// TIA Portal project "durum_grafigi_1" (V18)

(* hardware
DEVICE "S7-1200 station_1"  S7-1200 Station
   slot 0: "Rack_0"  S7-1200 Rack  Rack  V1.0
   slot 1: "PLC_1"  CPU 1214C DC/DC/DC  6ES7 214-1AG40-0XB0  V4.6
*)

// ===== PLC "PLC_1"  CPU 1214C DC/DC/DC =====

VAR_GLOBAL   // PLC tag table "Default tag table"
   "BAŞLAT" AT %I0.0 : Bool;
   "seviye_1_S1" AT %I0.1 : Bool;
   "seviye_2_S2" AT %I0.2 : Bool;
   "seviye_3_S3" AT %I0.3 : Bool;
   "ısı_sensoru_S4" AT %I0.4 : Bool;
   "valf_1" AT %Q0.1 : Bool;
   "valf_2" AT %Q0.2 : Bool;
   "valf_3" AT %Q0.3 : Bool;
   "ısıtıcı" AT %Q0.4 : Bool;
   "karıştırıcı" AT %Q0.5 : Bool;
   "System_Byte" AT %MB80 : Byte;
   "FirstScan" AT %M80.0 : Bool;
   "DiagStatusUptade" AT %M80.1 : Bool;
   "AlwaysTRUE" AT %M80.2 : Bool;
   "AlwaysFALSE" AT %M80.3 : Bool;
   "DURUM_0" AT %M30.0 : Bool;
   "DURUM_1" AT %M30.1 : Bool;
   "DURUM_2" AT %M30.2 : Bool;
   "DURUM_3" AT %M30.3 : Bool;
   "DURUM_4" AT %M30.4 : Bool;
END_VAR

ORGANIZATION_BLOCK "Main"   // OB1, LAD, ProgramCycle
TITLE = "Main Program Sweep (Cycle)"
{ S7_Optimized_Access := 'TRUE' }
VERSION : 0.1
   VAR_INPUT
      Initial_Call : Bool;   // Initial call of this OB
      Remanence : Bool;   // =True, if remanent data are available
   END_VAR
BEGIN

REGION Network 1: DURUM_0
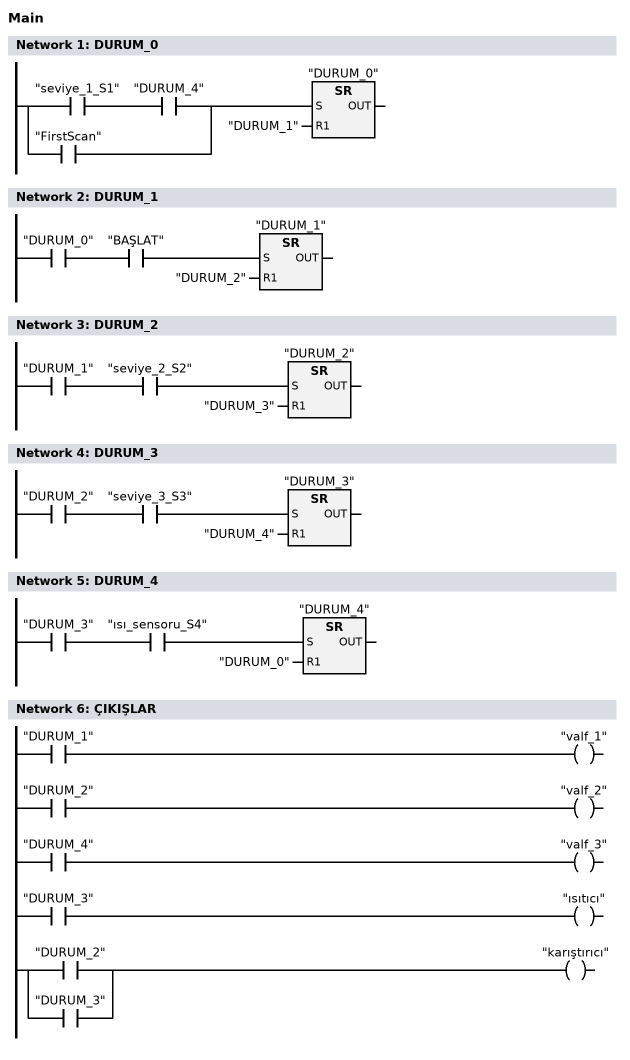
   RUNG wire#powerrail
      Contact( "seviye_1_S1" )
      Contact( "DURUM_4" )
      wire#w1
      S_SR(operand := "DURUM_0", r1 := "DURUM_1")
   END_RUNG
   RUNG wire#powerrail
      Contact( "FirstScan" )
   END_RUNG wire#w1
   // the same network as SCL:
   IF ("seviye_1_S1" AND "DURUM_4") OR "FirstScan" THEN
       "DURUM_0" := TRUE;   // SR flip-flop
   END_IF;
   IF "DURUM_1" THEN "DURUM_0" := FALSE; END_IF;
END_REGION

REGION Network 2: DURUM_1
   RUNG wire#powerrail
      Contact( "DURUM_0" )
      Contact( "BAŞLAT" )
      S_SR(operand := "DURUM_1", r1 := "DURUM_2")
   END_RUNG
   // the same network as SCL:
   IF "DURUM_0" AND "BAŞLAT" THEN
       "DURUM_1" := TRUE;   // SR flip-flop
   END_IF;
   IF "DURUM_2" THEN "DURUM_1" := FALSE; END_IF;
END_REGION

REGION Network 3: DURUM_2
   RUNG wire#powerrail
      Contact( "DURUM_1" )
      Contact( "seviye_2_S2" )
      S_SR(operand := "DURUM_2", r1 := "DURUM_3")
   END_RUNG
   // the same network as SCL:
   IF "DURUM_1" AND "seviye_2_S2" THEN
       "DURUM_2" := TRUE;   // SR flip-flop
   END_IF;
   IF "DURUM_3" THEN "DURUM_2" := FALSE; END_IF;
END_REGION

REGION Network 4: DURUM_3
   RUNG wire#powerrail
      Contact( "DURUM_2" )
      Contact( "seviye_3_S3" )
      S_SR(operand := "DURUM_3", r1 := "DURUM_4")
   END_RUNG
   // the same network as SCL:
   IF "DURUM_2" AND "seviye_3_S3" THEN
       "DURUM_3" := TRUE;   // SR flip-flop
   END_IF;
   IF "DURUM_4" THEN "DURUM_3" := FALSE; END_IF;
END_REGION

REGION Network 5: DURUM_4
   RUNG wire#powerrail
      Contact( "DURUM_3" )
      Contact( "ısı_sensoru_S4" )
      S_SR(operand := "DURUM_4", r1 := "DURUM_0")
   END_RUNG
   // the same network as SCL:
   IF "DURUM_3" AND "ısı_sensoru_S4" THEN
       "DURUM_4" := TRUE;   // SR flip-flop
   END_IF;
   IF "DURUM_0" THEN "DURUM_4" := FALSE; END_IF;
END_REGION

REGION Network 6: ÇIKIŞLAR
   RUNG wire#powerrail
      Contact( "DURUM_1" )
      Coil( "valf_1" )
   END_RUNG
   RUNG wire#powerrail
      Contact( "DURUM_2" )
      Coil( "valf_2" )
   END_RUNG
   RUNG wire#powerrail
      Contact( "DURUM_4" )
      Coil( "valf_3" )
   END_RUNG
   RUNG wire#powerrail
      Contact( "DURUM_3" )
      Coil( "ısıtıcı" )
   END_RUNG
   RUNG wire#powerrail
      Contact( "DURUM_2" )
      wire#w1
      Coil( "karıştırıcı" )
   END_RUNG
   RUNG wire#powerrail
      Contact( "DURUM_3" )
   END_RUNG wire#w1
   // the same network as SCL:
   "valf_1" := "DURUM_1";
   "valf_2" := "DURUM_2";
   "valf_3" := "DURUM_4";
   "ısıtıcı" := "DURUM_3";
   "karıştırıcı" := "DURUM_2" OR "DURUM_3";
END_REGION
END_ORGANIZATION_BLOCK